(* IEC 61131-3 sources: RL_MAR/experiments/comparison/autoplc/results/qwen3.5-9b_20260511_180311/med_58, 1 file *)

(* ---- med_58_1.st ---- *)
FUNCTION_BLOCK FB_ThresholdAccumulator
VAR_INPUT
i : INT;
END_VAR
VAR_OUTPUT
o : INT;
END_VAR
VAR
s1 : INT;
END_VAR

s1 := 0;
IF i > 0 THEN
s1 := s1 + i;
END_IF;
IF s1 = 42 THEN
s1 := s1 + 8000;
END_IF;
IF s1 < 0 THEN
o := 0;
ELSE
o := s1;
END_IF;
END_FUNCTION_BLOCK
